PROGRAM POU_DT01_EnableDriveTrain
VAR
	
	EnableDriveTrain 		: BOOL;
	
	fbLeftPower 			: MC_Power;
	LeftMotorEnabled		: BOOL;
	
	fbRightPower 			: MC_Power;
	RightMotorEnabled 		: BOOL;
	
END_VAR

EnableDriveTrain 			:= TRUE;

fbLeftPower(
	Axis					:= LeftMotor,
	Enable					:= EnableDriveTrain,
	Enable_Positive			:= TRUE,
	Status					=> LeftMotorEnabled);
	
fbRightPower(
	Axis					:= RightMotor,
	Enable					:= EnableDriveTrain,
	Enable_Positive			:= TRUE,
	Status					=> RightMotorEnabled);
	
IF LeftMotorEnabled AND RightMotorEnabled THEN
	
	DriveTrainEnabled 		:= TRUE;
	
ELSE
	
	DriveTrainEnabled 		:= FALSE;
	
END_IF

END_PROGRAM

(* stored: Version 1.1.0.1, ProductVersion 3.1.4022.7
   POU POU_DT01_EnableDriveTrain: Id {12442c86-3e4f-4aa0-b072-33d0a6e585a2}, SpecialFunc None *)
